Universal Robots PolyScope program: calibration_test_new.urp

Program calibration_test_new (installation=default directory=/programs/HandEyeCalibration createdIn=3.10.1.76190 lastSavedIn=5.10.0.106288 robotSerialNumber=20185500256)
Calibrated DH parameters: a=[0.000163, -0.146131, -0.38577, 0.000126, -0.000021, 0]; d=[0.161954, 188.306531, -157.478086, -30.695088, 0.099716, 0.099628]; alpha=[1.569701, -0.00212, 0.002263, 1.570438, -1.570123, 0]; deltaTheta=[0, -1.219859, 7.681919, -0.178877, -0.000001, 0]
BeforeStart
  calib_server := rpc_factory("xmlrpc", "http://192.168.1.119:10000")
Robot Program (runOnlyOnce=true)
  tcp_pose := get_actual_tcp_pose()
  board_pose := calib_server.test_extrinsic_calibration(tcp_pose)
  SuppressedNode
    board_pose := calib_server.test_extrinsic_calibration()
  init_board_pose := board_pose
  Script: board_pose[3]=tcp_pose[3]
  Script: board_pose[4]=tcp_pose[4]
  Script: board_pose[5]=tcp_pose[5]
  Script: board_pose[2]=board_pose[2]+0.01
  Popup Error (haltProgram=true message=debug stop inputType=Text)
  MoveL speed 250 mm/s, acceleration 1200 mm/s^2 (useActiveTCP=true) feature=Base
    Waypoint Waypoint (Variable): variable=board_pose
